TYPE Vec7di : ARRAY[1..7] OF DINT; END_TYPE

(* stored: Version 1.1.0.1, ProductVersion 3.1.4024.11
   DUT Vec7di: Id {516389f9-79e7-4ce5-80e0-ee6d29d0909c} *)
